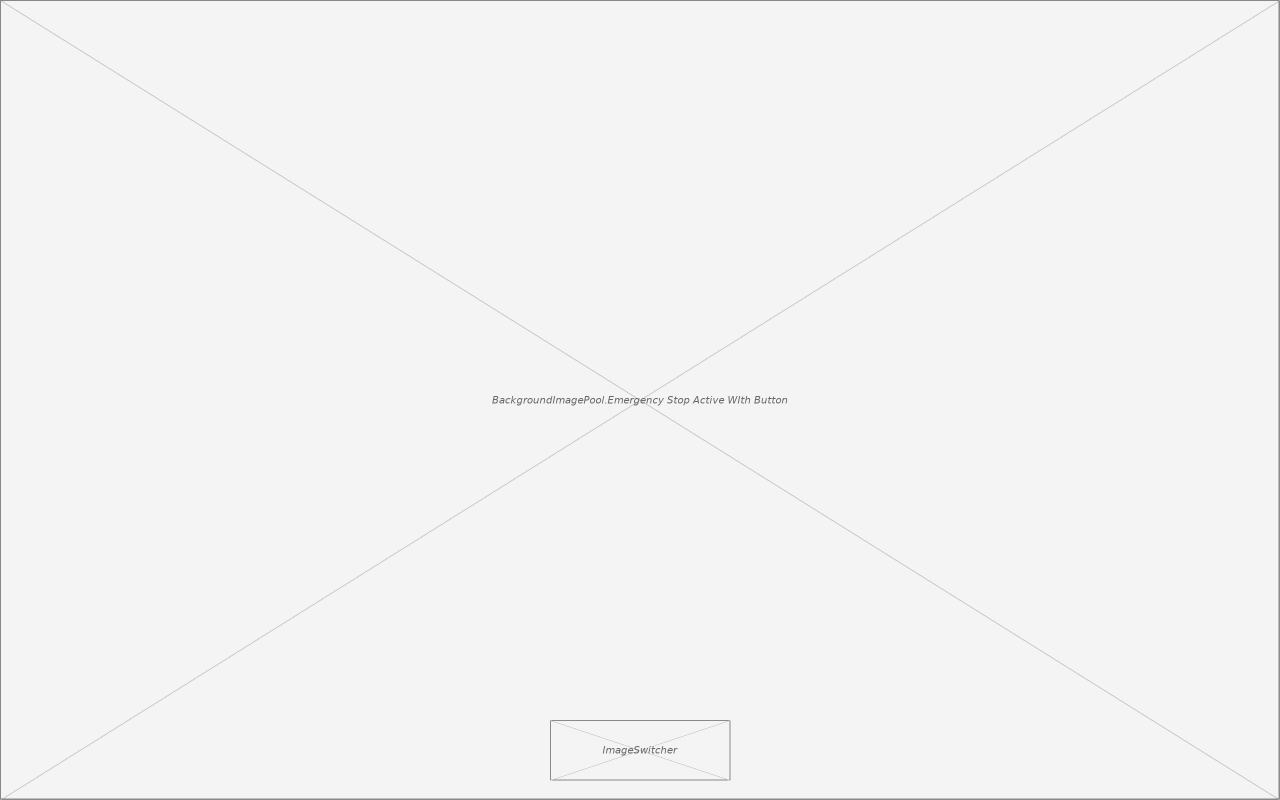
VISUALIZATION BackgroundWithBorder  // 1280x800, background image BackGroundImagePool_SVG.Background_Bottom
VAR_IN_OUT
	bCmdSettings 	: BOOL ; // to settings screen command
	bHideEstop		: BOOL ; // Hide Estop screen
	bDisableSettings: BOOL ; // Disable settings button
END_VAR
    Image (0,0 1280x800), invisible if: bHideEstop, input disabled if: bHideEstop, image: BackgroundImagePool.Emergency Stop Active WIth Button
    ImageSwitcher (550,720 180x60), variable: bCmdSettings, input disabled if: bDisableSettings, background image: Buttons_SVG.Home-Settings Switch Pushed, image: Buttons_SVG.Home Settings switch, behaviour: TOGGLE
        p3148411668: Buttons_SVG.Home-Settings Switch Pushed
END_VISUALIZATION

(* stored: Version 1.1.0.1, ProductVersion 3.1.4024.5
   Visu BackgroundWithBorder: Id {80a01c00-7e95-43c6-ba37-e4848c79e10a} *)
